FUNCTION_BLOCK CHASSIS_GENERATOR
  {SET_ATTRIBUTE(OpcUa, DEVICE.SENSOR)}
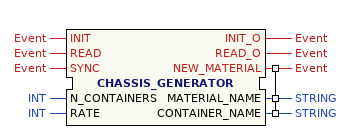
  EVENT_INPUT
    INIT;
    READ;
    SYNC;
  END_EVENT
  EVENT_OUTPUT
    INIT_O;
    READ_O;
    NEW_MATERIAL WITH MATERIAL_NAME, CONTAINER_NAME;
  END_EVENT
  VAR_INPUT
    N_CONTAINERS : INT; {SET_ATTRIBUTE(OpcUa, Constant)}
    RATE : INT; {SET_ATTRIBUTE(OpcUa, Constant)}
  END_VAR
  VAR_OUTPUT
    MATERIAL_NAME : STRING; {SET_ATTRIBUTE(OpcUa, Variable)}
    CONTAINER_NAME : STRING; {SET_ATTRIBUTE(OpcUa, Variable)}
  END_VAR
END_FUNCTION_BLOCK
